TYPE ST_MCHMIMachineControl_HMI :
STRUCT
	bZmienna : BOOL;
END_STRUCT
END_TYPE

(* stored: Version 1.1.0.1
   DUT ST_MCHMIMachineControl_HMI: Id {009353af-bf5e-0475-1b5c-fcccc8c8912e} *)
